INTERFACE I_Handler

METHOD handleRequest : BOOL
VAR_INPUT
	in_sRequest		: STRING;
END_VAR
END_METHOD

END_INTERFACE

(* stored: Version 1.1.0.1
   Itf I_Handler: Id {cc386116-5f2e-4e00-a127-9f41f328216d}
   Method handleRequest: Id {61fe22be-00f2-4ee8-84a9-7537e79d74a2} *)
